PROGRAM MAIN
VAR
END_VAR

END_PROGRAM

(* stored: Version 1.1.0.1
   POU MAIN: Id {320df1f8-468e-46a8-b990-e02f16a957b9} *)
